TYPE LREAL_Ext :
STRUCT
    Value       : LREAL;
    Permission  : DUT_Permission;
    bWrite      : BOOL;
    bBusy       : BOOL;
    bDone       : BOOL;
    bError      : BOOL;
END_STRUCT
END_TYPE

(* stored: Version 1.1.0.1, ProductVersion 3.1.4024.0
   DUT LREAL_Ext: Id {cb404dc4-8fef-404f-b5c4-416d65acd4ac} *)
